Yaskawa INFORM job: SR-ARC-1.JBI

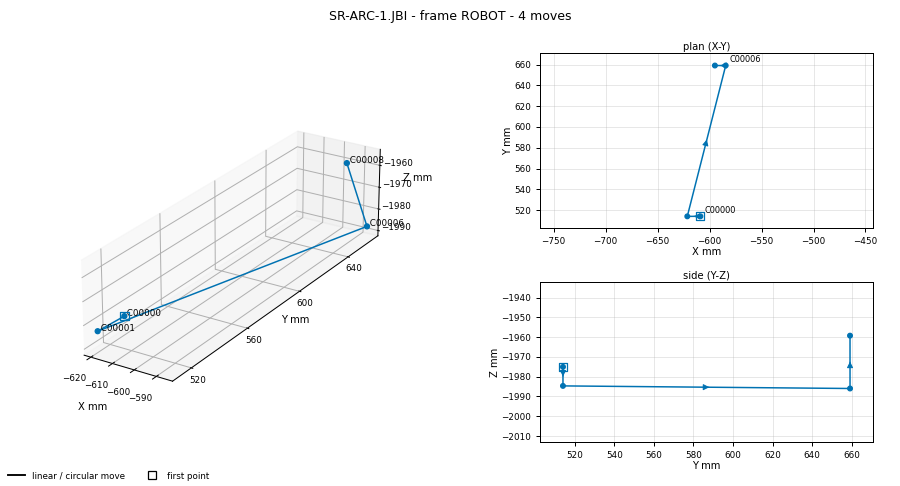
[picture p0: tool path of SR-ARC-1.JBI in frame ROBOT, 4 of 4 moves have a stored position in this frame; points joined in program order, loops and branches not executed]
/JOB
//NAME SR-ARC-1
///FOLDERNAME KRIS-SCIANA
//POS
///NPOS 9,6,0,1,0,0
///TOOL 0
///POSTYPE ROBOT
///RECTAN
///RCONF 0,0,0,0,0,0,0,0,0,0,0,0,0,0,0,0,0,0,0,0,0,0,0,0
C00000=-608.802,514.039,-1975.052,38.7850,-7.0699,82.9798
C00001=-621.415,514.030,-1984.662,38.7838,-7.0702,82.9805
///RCONF 0,0,0,0,1,0,0,0,0,0,0,0,0,0,0,0,0,0,0,0,0,0,0,0
C00002=-488.132,854.979,-1705.398,46.8018,1.8788,92.9494
C00003=-488.124,698.165,-1705.412,46.8005,1.8783,92.9506
C00004=-488.132,854.979,-1705.398,46.8018,1.8788,92.9494
///RCONF 0,0,0,0,0,0,0,0,0,0,0,0,0,0,0,0,0,0,0,0,0,0,0,0
C00005=-621.414,514.030,-1984.663,38.7842,-7.0696,82.9798
///RCONF 1,0,0,0,0,0,0,0,0,0,0,0,0,0,0,0,0,0,0,0,0,0,0,0
C00006=-584.463,659.112,-1985.972,37.1034,-7.5914,83.4049
///RCONF 0,0,0,0,1,0,0,0,0,0,0,0,0,0,0,0,0,0,0,0,0,0,0,0
C00007=-491.189,986.905,-1705.150,46.8017,1.8819,92.9474
///RCONF 1,0,0,0,0,0,0,0,0,0,0,0,0,0,0,0,0,0,0,0,0,0,0,0
C00008=-594.856,659.103,-1959.262,37.1033,-7.5909,83.4047
///RCONF 0,0,0,0,0,0,0,0,0,0,0,0,0,0,0,0,0,0,0,0,0,0,0,0
BC00000=2499.952,179.071,1196.539
BC00001=2499.952,179.071,1196.539
BC00002=2499.952,179.071,1196.539
BC00003=2499.952,179.071,1196.539
BC00004=2277.976,6088.070,599.815
BC00005=2499.952,179.071,1196.539
///POSTYPE BASE
P00070=2.449,-18.318,2.615,0.0000,0.0000,0.0000
//INST
///DATE 2023/12/20 15:47
///ATTR SC,RW,RJ
////FRAME ROBOT
///GROUP1 RB1,BS1
NOP
MOVL C00000 BC00000 V=150.0
MOVL C00001 BC00001 V=75.0
COMM MACRO1 MJ#(7) ARGFB000 ARGF1 ARGFC00002 ARGFC00003 ARGF1 ARGF70 ARGF4020 ARGF200 ARGF70
COMM PAUSE IF B001=0
COMM MACRO1 MJ#(8) ARGFB000 ARGFP070 ARGFC00004 ARGF1 ARGF500.0 ARGF71 ARGF4020
COMM PAUSE IF B001=0
COMM ARCON
MACRO1 MJ#(5) ARGFB000 ARGF1 ARGF450 ARGFC00005 ARGFBC00002 ARGF4020
MOVL C00006 BC00003 V=16.7
COMM MACRO1 MJ#(9) ARGFB000 ARGF1
COMM MOVL C00007 BC00004 V=16.7
MACRO1 MJ#(3) ARGFB000
COMM ARCOF
SFTOF
MOVL C00008 BC00005 V=75.0
END
